FUNCTION_BLOCK FB_Functions
VAR_INPUT
END_VAR
VAR_OUTPUT
END_VAR
VAR
END_VAR

{attribute 'TcRpcEnable'}
METHOD M_EnableAxis : BOOL
VAR_INPUT
	axisID : UINT;
	loopID : UINT;
END_VAR
Main.AxisPower(Axis:=Main.Axis[axisID][loopID],Enable:=TRUE,Enable_Positive:=TRUE,Enable_Negative:=TRUE); 

RETURN;
END_METHOD

{attribute 'TcRpcEnable'}
METHOD M_MoveAbsolute : BOOL
VAR_INPUT
	axisID : UINT;
	loopID : UINT;
	position : UINT;
	velocity : UINT;
END_VAR
Main.AxisPower(Axis:=Main.Axis[axisID][loopID],Enable:=TRUE,Enable_Positive:=TRUE,Enable_Negative:=TRUE); 

WHILE Main.Axis[axisID][loopID].Status.Operational = FALSE DO
	Main.MoveAbsolute(Axis:=Main.Axis[axisID][loopID],Execute:=FALSE);
END_WHILE

Main.MoveAbsolute(Axis:=Main.Axis[axisID][loopID],Execute:=FALSE);
Main.Reset(Axis:=Main.Axis[axisID][loopID],Execute:=FALSE);
			
Main.MoveAbsolute(Axis:=main.Axis[axisID][loopID],Position:=position,Velocity:=velocity);
					
Main.MoveAbsolute(Axis:=Main.Axis[axisID][loopID],Execute:=TRUE);

Main.MoveAbsolute(Axis:=Main.Axis[axisID][loopID],Execute:=FALSE);

RETURN;
END_METHOD

{attribute 'TcRpcEnable'}
METHOD M_MoveRelative : BOOL
VAR_INPUT
	axisID : UINT;
	loopID : UINT;
	position : UINT;
	velocity : UINT;
END_VAR
Main.AxisPower(Axis:=Main.Axis[axisID][loopID],Enable:=TRUE,Enable_Positive:=TRUE,Enable_Negative:=TRUE); 

WHILE Main.Axis[axisID][loopID].Status.Operational = FALSE DO
	Main.MoveRelative(Axis:=Main.Axis[axisID][loopID],Execute:=FALSE);
END_WHILE

Main.MoveRelative(Axis:=Main.Axis[axisID][loopID],Execute:=FALSE);
Main.Reset(Axis:=Main.Axis[axisID][loopID],Execute:=FALSE);
			
Main.MoveRelative(Axis:=Main.Axis[axisID][loopID],Distance:=position,Velocity:=velocity);
					
Main.MoveRelative(Axis:=Main.Axis[axisID][loopID],Execute:=TRUE);

Main.MoveRelative(Axis:=Main.Axis[axisID][loopID],Execute:=FALSE);

RETURN;
END_METHOD

{attribute 'TcRpcEnable'}
METHOD M_ReadActiveLoop : UINT
VAR_INPUT
	axisID : UINT;
END_VAR
VAR_OUTPUT
	loopID : UINT;
END_VAR
loopID := Main.Axis[axisID][0].NcToPlc.ActiveControlLoopIndex;

RETURN;
END_METHOD

{attribute 'TcRpcEnable'}
METHOD M_ReadAxisParameters : LREAL
VAR_INPUT
	axisID : UINT;
	loopID : UINT;
END_VAR
VAR_OUTPUT
	maxVelocity : LREAL;
	maxAcceleration : LREAL;
	defaultAcceleration : LREAL;
	defaultJerk : LREAL;
	homingVelocity : LREAL;
	manualVelocityFast : LREAL;
	manualVelocitySlow : LREAL;
	jogIncrement : LREAL;
END_VAR
// Axis Max Velocity
Main.ReadParameter(Axis:=Main.Axis[axisID][loopID],ParameterNumber:=MC_AxisParameter.AxisMaxVelocity);
Main.ReadParameter(Axis:=Main.Axis[axisID][loopID],Enable:=TRUE);
WHILE Main.ReadParameter.Busy DO
	Main.ReadParameter(Axis:=Main.Axis[axisID][loopID],Enable:=FALSE);
END_WHILE
maxVelocity := Main.ReadParameter.Value;


// Axis Max Acceleration
Main.ReadParameter(Axis:=Main.Axis[axisID][loopID],ParameterNumber:=MC_AxisParameter.AxisMaximumAcceleration);
Main.ReadParameter(Axis:=Main.Axis[axisID][loopID],Enable:=TRUE);
WHILE Main.ReadParameter.Busy DO
	Main.ReadParameter(Axis:=Main.Axis[axisID][loopID],Enable:=FALSE);
END_WHILE
maxAcceleration := Main.ReadParameter.Value;


//Axis Default Acceleration
Main.ReadParameter(Axis:=Main.Axis[axisID][loopID],ParameterNumber:=MC_AxisParameter.AxisAcc);
Main.ReadParameter(Axis:=Main.Axis[axisID][loopID],Enable:=TRUE);
WHILE Main.ReadParameter.Busy DO
	Main.ReadParameter(Axis:=Main.Axis[axisID][loopID],Enable:=FALSE);
END_WHILE
defaultAcceleration := Main.ReadParameter.Value;


//Axis Default Jerk
Main.ReadParameter(Axis:=Main.Axis[axisID][loopID],ParameterNumber:=MC_AxisParameter.AxisJerk);
Main.ReadParameter(Axis:=Main.Axis[axisID][loopID],Enable:=TRUE);
WHILE Main.ReadParameter.Busy DO
	Main.ReadParameter(Axis:=Main.Axis[axisID][loopID],Enable:=FALSE);
END_WHILE
defaultJerk := Main.ReadParameter.Value;


//Axis Homing Velocity +ve direction
Main.ReadParameter(Axis:=Main.Axis[axisID][loopID],ParameterNumber:=MC_AxisParameter.AxisCalibrationVelocityForward);
Main.ReadParameter(Axis:=Main.Axis[axisID][loopID],Enable:=TRUE);
WHILE Main.ReadParameter.Busy DO
	Main.ReadParameter(Axis:=Main.Axis[axisID][loopID],Enable:=FALSE);
END_WHILE
homingVelocity := Main.ReadParameter.Value;


//Axis Manual Velocity (Fast)
Main.ReadParameter(Axis:=Main.Axis[axisID][loopID],ParameterNumber:=MC_AxisParameter.AxisManualVelocityFast);
Main.ReadParameter(Axis:=Main.Axis[axisID][loopID],Enable:=TRUE);
WHILE Main.ReadParameter.Busy DO
	Main.ReadParameter(Axis:=Main.Axis[axisID][loopID],Enable:=FALSE);
END_WHILE
manualVelocityFast := Main.ReadParameter.Value;


//Axis Manual Velocity (Slow)
Main.ReadParameter(Axis:=Main.Axis[axisID][loopID],ParameterNumber:=MC_AxisParameter.AxisManualVelocitySlow);
Main.ReadParameter(Axis:=Main.Axis[axisID][loopID],Enable:=TRUE);
WHILE Main.ReadParameter.Busy DO
	Main.ReadParameter(Axis:=Main.Axis[axisID][loopID],Enable:=FALSE);
END_WHILE
manualVelocitySlow := Main.ReadParameter.Value;


//Axis Jog Increment +ve Direction
Main.ReadParameter(Axis:=Main.Axis[axisID][loopID],ParameterNumber:=MC_AxisParameter.AxisJogIncrementForward);
Main.ReadParameter(Axis:=Main.Axis[axisID][loopID],Enable:=TRUE);
WHILE Main.ReadParameter.Busy DO
	Main.ReadParameter(Axis:=Main.Axis[axisID][loopID],Enable:=FALSE);
END_WHILE
jogIncrement := Main.ReadParameter.Value;

RETURN;
END_METHOD

{attribute 'TcRpcEnable'}
METHOD M_ReadEncoderParameters : UINT
VAR_INPUT
	axisID : UINT;
	loopID : UINT;
END_VAR
VAR_OUTPUT
	invertEncoderDirection : BOOL;
	scalingFactorNumerator : LREAL;
	scalingFactorDenominator : LREAL;
	encoderOffset : LREAL;
	encoderMask : LREAL;
END_VAR
// Invert Encoder Direction
Main.ReadBoolParameter(Axis:=Main.Axis[axisID][loopID],ParameterNumber:=MC_AxisParameter.AxisEncoderDirectionInverse);
Main.ReadBoolParameter(Axis:=Main.Axis[axisID][loopID],Enable:=TRUE);
WHILE Main.ReadParameter.Busy DO
	Main.ReadBoolParameter(Axis:=Main.Axis[axisID][loopID],Enable:=FALSE);
END_WHILE
invertEncoderDirection := Main.ReadBoolParameter.Value;


// Encoder Scaling Factor Numerator
Main.ReadParameter(Axis:=Main.Axis[axisID][loopID],ParameterNumber:=MC_AxisParameter.AxisEncoderScalingNumerator);
Main.ReadParameter(Axis:=Main.Axis[axisID][loopID],Enable:=TRUE);
WHILE Main.ReadParameter.Busy DO
	Main.ReadParameter(Axis:=Main.Axis[axisID][loopID],Enable:=FALSE);
END_WHILE
scalingFactorNumerator := Main.ReadParameter.Value;


// Encoder Scaling Factor Denominator
Main.ReadParameter(Axis:=Main.Axis[axisID][loopID],ParameterNumber:=MC_AxisParameter.AxisEncoderScalingDenominator);
Main.ReadParameter(Axis:=Main.Axis[axisID][loopID],Enable:=TRUE);
WHILE Main.ReadParameter.Busy DO
	Main.ReadParameter(Axis:=Main.Axis[axisID][loopID],Enable:=FALSE);
END_WHILE
scalingFactorDenominator := Main.ReadParameter.Value;


// Encoder Offset
Main.ReadParameter(Axis:=Main.Axis[axisID][loopID],ParameterNumber:=MC_AxisParameter.AxisEncoderOffset);
Main.ReadParameter(Axis:=Main.Axis[axisID][loopID],Enable:=TRUE);
WHILE Main.ReadParameter.Busy DO
	Main.ReadParameter(Axis:=Main.Axis[axisID][loopID],Enable:=FALSE);
END_WHILE
encoderOffset := Main.ReadParameter.Value;


// Encoder Mask
Main.ReadParameter(Axis:=Main.Axis[axisID][loopID],ParameterNumber:=MC_AxisParameter.AxisEncoderMask);
Main.ReadParameter(Axis:=Main.Axis[axisID][loopID],Enable:=TRUE);
WHILE Main.ReadParameter.Busy DO
	Main.ReadParameter(Axis:=Main.Axis[axisID][loopID],Enable:=FALSE);
END_WHILE
encoderMask := Main.ReadParameter.Value;


RETURN;
END_METHOD

{attribute 'TcRpcEnable'}
METHOD M_SetActiveEncoder : BOOL
VAR_INPUT
	axisID : UINT;
	loopID : UINT;
END_VAR
Main.SetControlLoop(Axis:=Main.Axis[axisID][loopID],Execute:=FALSE,SelectType:=E_SelectControlLoopType.SelectControlLoopType_Standard,EncoderIndex:=loopID);
Main.SetControlLoop(Axis:=Main.Axis[axisID][loopID],Execute:=TRUE);
WHILE (Main.SetControlLoop.Done=FALSE) DO
	Main.SetControlLoop(Axis:=Main.Axis[axisID][loopID],Execute:=FALSE);
END_WHILE

RETURN;
END_METHOD

{attribute 'TcRpcEnable'}
METHOD M_WriteAxisParameters : BOOL
VAR_INPUT
	axisID: UINT;
	loopID: UINT;
	maxVelocity : UINT;
	maxAcceleration : UINT;
	defaultAcceleration : UINT;
	defaultJerk : UINT;
	homingVelocity : UINT;
	manualVelocityFast : UINT;
	manualVelocitySlow : UINT;
	jogIncrement : UINT;
END_VAR
// Axis Max Velocity
Main.WriteParameter(Axis:=Main.Axis[axisID][loopID],ParameterNumber:=MC_AxisParameter.AxisMaxVelocity,Value:=maxVelocity);
Main.WriteParameter(Axis:=Main.Axis[axisID][loopID],Execute:=TRUE);
WHILE (Main.WriteParameter.Busy) DO
	Main.WriteParameter(Axis:=Main.Axis[axisID][loopID],Execute:=FALSE);
END_WHILE

// Axis Max Acceleration
Main.WriteParameter(Axis:=Main.Axis[axisID][loopID],ParameterNumber:=MC_AxisParameter.AxisMaximumAcceleration,Value:=maxAcceleration);
Main.WriteParameter(Axis:=Main.Axis[axisID][loopID],Execute:=TRUE);
WHILE (Main.WriteParameter.Busy) DO
	Main.WriteParameter(Axis:=Main.Axis[axisID][loopID],Execute:=FALSE);
END_WHILE

//Axis Max Deceleration
Main.WriteParameter(Axis:=Main.Axis[axisID][loopID],ParameterNumber:=MC_AxisParameter.AxisMaximumDeceleration,Value:=maxAcceleration);
Main.WriteParameter(Axis:=Main.Axis[axisID][loopID],Execute:=TRUE);
WHILE (Main.WriteParameter.Busy) DO
	Main.WriteParameter(Axis:=Main.Axis[axisID][loopID],Execute:=FALSE);
END_WHILE

//Axis Default Acceleration
Main.WriteParameter(Axis:=Main.Axis[axisID][loopID],ParameterNumber:=MC_AxisParameter.AxisAcc,Value:=defaultAcceleration);
Main.WriteParameter(Axis:=Main.Axis[axisID][loopID],Execute:=TRUE);
WHILE (Main.WriteParameter.Busy) DO
	Main.WriteParameter(Axis:=Main.Axis[axisID][loopID],Execute:=FALSE);
END_WHILE

//Axis Default Deceleration
Main.WriteParameter(Axis:=Main.Axis[axisID][loopID],ParameterNumber:=MC_AxisParameter.AxisDec,Value:=defaultAcceleration);
Main.WriteParameter(Axis:=Main.Axis[axisID][loopID],Execute:=TRUE);
WHILE (Main.WriteParameter.Busy) DO
	Main.WriteParameter(Axis:=Main.Axis[axisID][loopID],Execute:=FALSE);
END_WHILE

//Axis Default Jerk
Main.WriteParameter(Axis:=Main.Axis[axisID][loopID],ParameterNumber:=MC_AxisParameter.AxisJerk,Value:=defaultJerk);
Main.WriteParameter(Axis:=Main.Axis[axisID][loopID],Execute:=TRUE);
WHILE (Main.WriteParameter.Busy) DO
	Main.WriteParameter(Axis:=Main.Axis[axisID][loopID],Execute:=FALSE);
END_WHILE

//Axis Homing Velocity +ve direction
Main.WriteParameter(Axis:=Main.Axis[axisID][loopID],ParameterNumber:=MC_AxisParameter.AxisCalibrationVelocityForward,Value:=homingVelocity);
Main.WriteParameter(Axis:=Main.Axis[axisID][loopID],Execute:=TRUE);
WHILE (Main.WriteParameter.Busy) DO
	Main.WriteParameter(Axis:=Main.Axis[axisID][loopID],Execute:=FALSE);
END_WHILE

//Axis Homing Velocity -ve Direction
Main.WriteParameter(Axis:=Main.Axis[axisID][loopID],ParameterNumber:=MC_AxisParameter.AxisCalibrationVelocityBackward,Value:=homingVelocity);
Main.WriteParameter(Axis:=Main.Axis[axisID][loopID],Execute:=TRUE);
WHILE (Main.WriteParameter.Busy) DO
	Main.WriteParameter(Axis:=Main.Axis[axisID][loopID],Execute:=FALSE);
END_WHILE

//Axis Manual Velocity (Fast)
Main.WriteParameter(Axis:=Main.Axis[axisID][loopID],ParameterNumber:=MC_AxisParameter.AxisManualVelocityFast,Value:=manualVelocityFast);
Main.WriteParameter(Axis:=Main.Axis[axisID][loopID],Execute:=TRUE);
WHILE (Main.WriteParameter.Busy) DO
	Main.WriteParameter(Axis:=Main.Axis[axisID][loopID],Execute:=FALSE);
END_WHILE

//Axis Manual Velocity (Slow)
Main.WriteParameter(Axis:=Main.Axis[axisID][loopID],ParameterNumber:=MC_AxisParameter.AxisManualVelocitySlow,Value:=manualVelocitySlow);
Main.WriteParameter(Axis:=Main.Axis[axisID][loopID],Execute:=TRUE);
WHILE (Main.WriteParameter.Busy) DO
	Main.WriteParameter(Axis:=Main.Axis[axisID][loopID],Execute:=FALSE);
END_WHILE

//Axis Jog Increment +ve Direction
Main.WriteParameter(Axis:=Main.Axis[axisID][loopID],ParameterNumber:=MC_AxisParameter.AxisJogIncrementForward,Value:=jogIncrement);
Main.WriteParameter(Axis:=Main.Axis[axisID][loopID],Execute:=TRUE);
WHILE (Main.WriteParameter.Busy) DO
	Main.WriteParameter(Axis:=Main.Axis[axisID][loopID],Execute:=FALSE);
END_WHILE

//Axis Jog Increment -ve Direction
Main.WriteParameter(Axis:=Main.Axis[axisID][loopID],ParameterNumber:=MC_AxisParameter.AxisJogIncrementBackward,Value:=jogIncrement);
Main.WriteParameter(Axis:=Main.Axis[axisID][loopID],Execute:=TRUE);
WHILE (Main.WriteParameter.Busy) DO
	Main.WriteParameter(Axis:=Main.Axis[axisID][loopID],Execute:=FALSE);
END_WHILE

RETURN;
END_METHOD

{attribute 'TcRpcEnable'}
METHOD M_WriteEncoderParameters : BOOL
VAR_INPUT
	axisID : UINT;
	loopID : UINT;
	//invertEncoderDirection : BOOL;
	scalingFactorNumerator : LREAL;
	scalingFactorDenominator : LREAL;
	encoderOffset : UINT;
	encoderMask : DINT;
END_VAR
// encoder direction inverse
//Main.WriteBoolParameter(Axis:=Main.Axis1[controlLoopID],ParameterNumber:=MC_AxisParameter.AxisEncoderDirectionInverse,Value:=invertEncoderDirection);
//Main.WriteBoolParameter(Axis:=Main.Axis1[controlLoopID],Execute:=TRUE);
//WHILE (Main.WriteBoolParameter.Busy) DO
//	Main.WriteParameter(Axis:=Main.Axis1[controlLoopID],Execute:=FALSE);
//END_WHILE

// Encoder scaling factor numerator
Main.WriteParameter(Axis:=Main.Axis[0][loopID],ParameterNumber:=MC_AxisParameter.AxisEncoderScalingNumerator,Value:=scalingFactorNumerator);
Main.WriteParameter(Axis:=Main.Axis[axisID][loopID],Execute:=TRUE);
WHILE (Main.WriteParameter.Busy) DO
	Main.WriteParameter(Axis:=Main.Axis[axisID][loopID],Execute:=FALSE);
END_WHILE

// Encoder scaling factor denominator
Main.WriteParameter(Axis:=Main.Axis[axisID][loopID],ParameterNumber:=MC_AxisParameter.AxisEncoderScalingDenominator,Value:=scalingFactorDenominator);
Main.WriteParameter(Axis:=Main.Axis[axisID][loopID],Execute:=TRUE);
WHILE (Main.WriteParameter.Busy) DO
	Main.WriteParameter(Axis:=Main.Axis[axisID][loopID],Execute:=FALSE);
END_WHILE

// Encoder offset
Main.WriteParameter(Axis:=Main.Axis[axisID][loopID],ParameterNumber:=MC_AxisParameter.AxisEncoderOffset,Value:=encoderOffset);
Main.WriteParameter(Axis:=Main.Axis[axisID][loopID],Execute:=TRUE);
WHILE (Main.WriteParameter.Busy) DO
	Main.WriteParameter(Axis:=Main.Axis[axisID][loopID],Execute:=FALSE);
END_WHILE

// Encoder Mask
Main.WriteParameter(Axis:=Main.Axis[axisID][loopID],ParameterNumber:=MC_AxisParameter.AxisEncoderMask,Value:=encoderMask);
Main.WriteParameter(Axis:=Main.Axis[axisID][loopID],Execute:=TRUE);
WHILE (Main.WriteParameter.Busy) DO
	Main.WriteParameter(Axis:=Main.Axis[axisID][loopID],Execute:=FALSE);
END_WHILE

RETURN;
END_METHOD

END_FUNCTION_BLOCK

(* stored: Version 1.1.0.1, ProductVersion 3.1.4024.12
   POU FB_Functions: Id {87e7f3b9-d9e3-4e1a-ad5e-3d4326ef9e7d}, SpecialFunc None
   Method M_EnableAxis: Id {a241beb0-66b2-4f66-a177-89d82c51ec16}
   Method M_MoveAbsolute: Id {21c8d92b-8bc3-49df-8463-a5f13171cc19}
   Method M_MoveRelative: Id {49a2a512-3e94-4879-b314-10353ec76639}
   Method M_ReadActiveLoop: Id {e51264ef-8758-4e07-9f48-0556be0a0f46}
   Method M_ReadAxisParameters: Id {b4b35217-25df-4f47-ab66-df6486a56b0b}
   Method M_ReadEncoderParameters: Id {36292ad9-d555-42b3-804e-9c81d4086bc8}
   Method M_SetActiveEncoder: Id {9a091db5-976f-4ff2-9331-531b0095b97c}
   Method M_WriteAxisParameters: Id {66fe626f-3ffa-44ff-b51a-f7cf0d645e56}
   Method M_WriteEncoderParameters: Id {75354755-7da6-4b6c-bdbd-b438e676dd36} *)
